PROGRAM AUTO_SCREWPICKUP
VAR
END_VAR

END_PROGRAM

(* stored: Version 1.1.0.1, ProductVersion 3.1.4022.18
   POU AUTO_SCREWPICKUP: Id {c4db5fdc-7d52-49e3-beb9-79bd9a3b7f44}, SpecialFunc None *)
